Yaskawa INFORM job: X2_29-32(-90,180).JBI

/JOB
//NAME X2_29-32(-90,180)
//POS
///NPOS 301,301,301,19,0,0
///TOOL 0
///POSTYPE PULSE
///PULSE
C00000=-2000,-95440,-72516,0,38121,0
C00001=80443,-95440,-72516,46202,38121,-50067
C00002=52411,-63190,-65629,41206,65263,-51508
C00003=73087,-23788,-54178,20049,70640,-39353
C00004=137855,-58890,-63164,-50426,57117,-3007
C00005=121629,-1819,-23267,-32035,72941,-16834
C00006=120935,3126,-16373,-32060,71231,-16611
C00007=120668,5150,-13541,-32087,70531,-16512
C00008=120826,7275,-11699,-32150,70554,-16454
C00009=120668,5150,-13541,-32087,70531,-16512
C00010=120649,6560,-12069,-32112,70369,-16472
C00011=120645,6560,-10825,-32251,69714,-16277
C00012=120649,6560,-12069,-32112,70369,-16472
C00013=120913,4529,-14922,-32082,71075,-16573
C00014=121602,-429,-21862,-32048,72802,-16805
C00015=120074,-1541,-23154,-10906,71264,-22392
C00016=120462,3262,-16191,-11181,69532,-22093
C00017=120612,5232,-13331,-11295,68818,-21971
C00018=120770,7357,-11488,-11363,68799,-21912
C00019=120612,5232,-13331,-11295,68818,-21971
C00020=120702,6360,-12382,-11332,68826,-21940
C00021=120699,6356,-11141,-11388,68075,-21868
C00022=120702,6360,-12382,-11332,68826,-21940
C00023=120555,4389,-15254,-11219,69547,-22062
C00024=120172,-412,-22245,-10944,71297,-22361
C00025=119941,-49108,-60020,-12756,52739,-20459
C00026=119789,-74783,-79746,-11606,60570,-21449
C00027=121427,-115493,-86071,971,23186,-13
C00028=103613,-33005,-61039,35202,65094,22685
C00029=118652,-1130,-18887,50959,75871,22344
C00030=120065,3095,-12579,50928,73991,22034
C00031=120612,5858,-10323,50783,73711,22168
C00032=120794,7716,-8707,50742,73586,22192
C00033=120612,6719,-9575,50786,73699,22162
C00034=120612,6754,-8612,50907,73330,21953
C00035=120612,6719,-9575,50786,73699,22162
C00036=120164,4326,-11494,50910,73914,22043
C00037=118762,92,-17836,50934,75798,22362
C00038=120082,-2017,-23568,21020,76850,12939
C00039=120471,2786,-16617,21041,75059,12760
C00040=120621,6055,-13261,21027,74660,12744
C00041=120866,7545,-11965,20950,74569,12818
C00042=120698,6523,-12855,21003,74632,12768
C00043=120698,6506,-12245,21039,74273,12705
C00044=120698,6523,-12855,21003,74632,12768
C00045=120547,3972,-15593,21018,75020,12781
C00046=120163,-831,-22574,20994,76828,12964
C00047=120068,-2141,-23641,4094,79360,-4817
C00048=120458,2664,-16692,4000,77538,-4745
C00049=120609,5664,-13523,3960,77123,-4708
C00050=120915,7025,-12341,3868,77081,-4605
C00051=120609,5664,-13523,3960,77123,-4708
C00052=120609,5646,-12752,3962,76640,-4725
C00053=120609,5664,-13523,3960,77123,-4708
C00054=120559,4206,-15421,3970,77544,-4711
C00055=120175,-595,-22406,4061,79389,-4780
C00056=120687,14555,-20541,8533,86827,-5332
C00057=120686,13734,-18343,8544,85071,-5452
C00058=120482,15241,-16931,8603,84997,-5522
C00059=120827,14092,-17818,8504,84929,-5415
C00060=120926,18700,-11185,23232,84202,11400
C00061=120686,12663,-14714,25421,80171,12532
C00062=120686,13236,-17122,25321,81784,12881
C00063=103613,-33005,-61039,35202,65094,22685
C00064=121427,-115493,-86071,971,23186,-13
C00065=119789,-74783,-79746,-11606,60570,-21449
C00066=119941,-49108,-60020,-12756,52739,-20459
C00067=120686,14191,-18554,-15918,76373,-21593
C00068=120686,13500,-16249,-16032,74665,-21366
C00069=120864,13188,-15327,-16153,73998,-21217
C00070=120686,13025,-15397,-16089,73932,-21265
C00071=120685,13123,3553,-58384,63482,-21536
C00072=120685,12978,2576,-58170,63769,-21763
C00073=120685,12646,-109,-57582,64586,-22394
C00074=118042,2280,-28025,-21530,77386,-23855
C00075=119941,-49108,-60020,-12756,52739,-20459
C00076=119789,-74783,-79746,-11606,60570,-21449
C00077=121427,-115493,-86071,971,23186,-13
C00078=103613,-33005,-61039,35202,65094,22685
C00079=134099,37874,13933,30657,62495,29160
C00080=134100,37847,15487,30911,61654,28907
C00081=131666,39479,18748,33791,61688,27713
C00082=133865,38968,17694,31358,61081,28616
C00083=133702,39552,25338,55816,81533,5296
C00084=134106,38448,23823,57095,83317,3747
C00085=130543,37529,20923,57393,86199,3579
C00086=127607,4606,-13504,21031,60979,-34641
C00087=124532,-28339,-37080,-2656,37858,-63256
C00088=80443,-95440,-72516,46202,38121,-50067
C00089=628,-74499,-67639,57475,89722,-72456
C00090=-3643,-76224,-106676,-19950,71810,-76872
C00091=57022,-39792,-97587,14580,73098,-62715
C00092=77894,6609,-39652,10081,68656,-55583
C00093=79326,8848,-34628,9340,66588,-55287
C00094=79882,9812,-32559,9051,65763,-55166
C00095=80655,11957,-30643,8578,65611,-54918
C00096=79882,9812,-32559,9051,65763,-55166
C00097=80541,11612,-30977,8647,65649,-54954
C00098=80539,10894,-29907,8717,64633,-55031
C00099=80541,11612,-30977,8647,65649,-54954
C00100=79996,10638,-33064,8931,66478,-55073
C00101=78593,8374,-38132,9661,68553,-55366
C00102=77879,6415,-39661,10096,68566,-55596
C00103=79312,8664,-34633,9354,66499,-55298
C00104=79868,9631,-32562,9065,65674,-55178
C00105=80642,11778,-30647,8592,65523,-54929
C00106=79868,9631,-32562,9065,65674,-55178
C00107=80486,11377,-31039,8686,65573,-54978
C00108=80483,10662,-29965,8757,64557,-55056
C00109=80486,11377,-31039,8686,65573,-54978
C00110=79940,10400,-33127,8971,66401,-55097
C00111=78534,8129,-38197,9702,68474,-55392
C00112=80648,1920,-43069,8432,68075,-54741
C00113=82055,4328,-37962,7677,66061,-54418
C00114=82600,5356,-35863,7382,65258,-54288
C00115=83359,7582,-33929,6913,65152,-54039
C00116=82600,5356,-35863,7382,65258,-54288
C00117=83222,7216,-34336,6994,65225,-54082
C00118=83219,6503,-33246,7053,64194,-54145
C00119=83222,7216,-34336,6994,65225,-54082
C00120=82688,6183,-36451,7284,66032,-54210
C00121=81310,3762,-41594,8027,68053,-54528
C00122=103257,-17880,-58539,-5534,67057,-47481
C00123=104214,-14456,-52937,-6200,65440,-47084
C00124=104581,-13049,-50655,-6463,64788,-46925
C00125=105090,-10289,-48529,-6776,64935,-46761
C00126=104581,-13049,-50655,-6463,64788,-46925
C00127=105018,-10709,-48980,-6727,64992,-46789
C00128=105013,-11445,-47840,-6782,63918,-46728
C00129=105018,-10709,-48980,-6727,64992,-46789
C00130=104661,-12103,-51269,-6469,65653,-46947
C00131=103731,-15489,-56889,-5817,67299,-47340
C00132=80233,11979,-33534,13378,69985,-55632
C00133=80229,10556,-31784,13533,68226,-55836
C00134=80227,10062,-31089,13596,67561,-55913
C00135=85904,3072,-37201,10254,66968,-54061
C00136=91588,-2653,-41861,6857,66347,-52204
C00137=101831,-9955,-47602,630,65696,-48799
C00138=101534,-9526,-48387,809,66398,-48894
C00139=100861,-7653,-49935,1203,68321,-49097
C00140=80300,11336,-32181,3939,63811,-54132
C00141=80297,10024,-30348,4003,62013,-54196
C00142=80296,9591,-29657,4027,61367,-54219
C00143=80356,9906,-29534,3997,61454,-54195
C00144=80338,10281,-30338,3972,62137,-54177
C00145=80341,11605,-32161,3909,63935,-54114
C00146=57022,-39792,-97587,14580,73098,-62715
C00147=628,-74499,-67639,57475,89722,-72456
C00148=628,-74499,-67639,57475,89722,-72456
C00149=616,-75233,-71189,57531,90735,-71761
C00150=-3643,-76224,-106674,-19950,71813,-76873
C00151=42730,11015,-70691,38334,96086,-2936
C00152=63606,9545,-60534,45336,92087,16638
C00153=78956,5069,-41799,36523,82652,30708
C00154=79715,8164,-36018,36343,80767,30358
C00155=80007,9457,-33651,36288,80012,30216
C00156=80417,12097,-31285,36126,79775,30292
C00157=80007,9457,-33651,36288,80012,30216
C00158=80344,11698,-31669,36153,79828,30282
C00159=80337,10939,-30633,36254,78993,30001
C00160=80344,11698,-31669,36153,79828,30282
C00161=80059,10405,-34052,36203,80590,30428
C00162=79319,7312,-39869,36371,82488,30786
C00163=78994,5332,-41692,36502,82694,30736
C00164=79751,8420,-35912,36322,80808,30385
C00165=80043,9710,-33546,36267,80051,30242
C00166=80452,12349,-31177,36105,79813,30317
C00167=80043,9710,-33546,36267,80051,30242
C00168=80378,11838,-31671,36133,79874,30310
C00169=80371,11075,-30637,36233,79039,30029
C00170=80378,11838,-31671,36133,79874,30310
C00171=80093,10547,-34052,36183,80637,30456
C00172=79355,7462,-39866,36352,82536,30815
C00173=79090,5824,-41546,36452,82791,30803
C00174=79842,8894,-35770,36272,80900,30451
C00175=80133,10177,-33405,36216,80142,30307
C00176=80539,12815,-31031,36055,79902,30380
C00177=80133,10177,-33405,36216,80142,30307
C00178=80467,12378,-31515,36079,79989,30382
C00179=80461,11606,-30490,36178,79153,30101
C00180=80467,12378,-31515,36079,79989,30382
C00181=80184,11095,-33894,36130,80753,30529
C00182=79450,8031,-39703,36300,82657,30890
C00183=79130,5997,-41490,36432,82820,30827
C00184=79881,9061,-35715,36251,80928,30474
C00185=80171,10342,-33350,36196,80169,30330
C00186=80577,12980,-30974,36035,79928,30403
C00187=80171,10342,-33350,36196,80169,30330
C00188=80499,12601,-31443,36059,80034,30409
C00189=80493,11826,-30422,36158,79199,30129
C00190=80499,12601,-31443,36059,80034,30409
C00191=80216,11321,-33822,36110,80799,30556
C00192=79484,8265,-39628,36281,82705,30918
C00193=80360,13355,-34008,31162,79863,31191
C00194=80358,11846,-32319,31320,78301,30757
C00195=80218,11485,-31511,31450,77760,30555
C00196=80458,11751,-31298,31342,77685,30622
C00197=80398,12063,-32232,31297,78337,30782
C00198=80400,13577,-33916,31139,79899,31215
C00199=80289,11819,-32883,40833,82428,30239
C00200=80286,10439,-31086,40975,81039,29694
C00201=80075,10175,-30147,41122,80582,29428
C00202=80234,9688,-30441,41065,80463,29445
C00203=80245,10226,-31168,40996,81011,29666
C00204=80248,11601,-32971,40853,82401,30212
C00205=66712,19655,-58640,43457,90055,24381
C00206=33423,17994,-60377,60627,102988,19600
C00207=628,-74499,-67639,57475,89722,77289
C00208=111516,-94989,-87682,11539,41033,8318
C00209=107125,-12532,-46236,32676,64375,10703
C00210=119952,37605,6162,31233,75137,17424
C00211=120511,42562,14108,31354,72919,17016
C00212=120728,44654,17433,31427,72005,16841
C00213=120598,46946,19889,31526,71766,16719
C00214=120728,44654,17433,31427,72005,16841
C00215=120690,45788,18679,31469,71861,16784
C00216=120687,45721,19851,31594,71213,16595
C00217=120690,45788,18679,31469,71861,16784
C00218=120474,43679,15324,31394,72783,16962
C00219=119917,38688,7316,31265,75018,17376
C00220=121235,29127,929,10497,72605,22385
C00221=120892,33963,8709,10768,70384,22067
C00222=120760,35995,11952,10883,69467,21936
C00223=120625,38237,14258,10956,69222,21864
C00224=120760,35995,11952,10883,69467,21936
C00225=120657,37146,13206,10937,69303,21884
C00226=120654,37124,14427,10991,68554,21813
C00227=120657,37146,13206,10937,69303,21884
C00228=120788,35099,9935,10821,70230,22016
C00229=121127,30229,2096,10548,72470,22335
C00230=114017,-48711,-62992,16459,47417,13874
C00231=111516,-94989,-87682,11539,41033,8318
C00232=135207,-75469,-94215,-36619,68365,-13249
C00233=122507,12852,-43627,-17515,100315,-22769
C00234=122731,-562,-19309,-51196,76332,-22742
C00235=121309,3590,-13049,-51151,74446,-22427
C00236=120759,5312,-10468,-51156,73690,-22291
C00237=120602,7442,-8613,-51127,73573,-22309
C00238=120759,5312,-10468,-51156,73690,-22291
C00239=120666,6547,-9361,-51143,73609,-22295
C00240=120662,6597,-8073,-51308,73115,-22013
C00241=120666,6547,-9361,-51143,73609,-22295
C00242=121212,4820,-11958,-51134,74367,-22434
C00243=122622,659,-18251,-51172,76257,-22758
C00244=122507,10859,-42333,-17402,98575,-22516
C00245=121302,-1391,-23074,-21379,77148,-13095
C00246=120901,3377,-16122,-21398,75339,-12912
C00247=120747,5333,-13267,-21416,74597,-12833
C00248=120590,7459,-11416,-21370,74514,-12875
C00249=120747,5333,-13267,-21416,74597,-12833
C00250=120673,6521,-12221,-21396,74547,-12851
C00251=120670,6504,-10992,-21468,73832,-12721
C00252=120673,6521,-12221,-21396,74547,-12851
C00253=120826,4563,-15090,-21376,75296,-12931
C00254=121222,-206,-22073,-21354,77121,-13119
C00255=121314,-1652,-23262,-4485,79740,4708
C00256=120913,3117,-16316,-4391,77900,4639
C00257=120758,5074,-13462,-4356,77144,4613
C00258=120601,7199,-11615,-4311,77090,4561
C00259=120758,5074,-13462,-4356,77144,4613
C00260=120661,6618,-12165,-4328,77134,4580
C00261=120658,6600,-10936,-4339,76370,4606
C00262=120661,6618,-12165,-4328,77134,4580
C00263=120814,4660,-15035,-4362,77900,4605
C00264=121209,-107,-22019,-4454,79763,4672
C00265=120687,46979,12625,-8958,83453,5452
C00266=120687,46939,12852,-8960,83294,5464
C00267=121610,47264,14210,-9230,82736,5807
C00268=120687,46849,13873,-8967,82635,5512
C00269=120687,46629,18284,-25995,77833,-12130
C00270=120687,46348,16793,-25935,78533,-12285
C00271=120687,46750,14296,-25811,80109,-12635
C00272=133650,-5326,-40947,-35821,67459,-4738
C00273=126605,-79487,-84548,-34660,58331,-13454
C00274=111516,-94989,-87682,11539,41033,8318
C00275=114017,-48711,-62992,16459,47417,13874
C00276=117875,8541,-26754,15356,68464,18868
C00277=120687,46680,12303,15684,74586,21239
C00278=120687,46183,14573,15804,72993,21028
C00279=120687,45847,15503,15862,72274,20933
C00280=120687,45820,15711,15860,72146,20914
C00281=120686,46430,31549,51889,62431,21622
C00282=120686,46225,30262,51616,62867,21897
C00283=120686,45862,27317,50999,63909,22538
C00284=117875,8541,-26754,15356,68464,18868
C00285=114017,-48711,-62992,16459,47417,13874
C00286=111516,-94989,-87682,11539,41033,8318
C00287=126605,-79487,-84548,-34660,58331,-13454
C00288=133650,-5326,-40947,-35821,67459,-4738
C00289=107292,16878,-7589,-30401,64778,-29950
C00290=107291,16671,-4858,-30829,63228,-29495
C00291=107592,16882,-3413,-31166,62662,-29196
C00292=107321,17068,-3230,-31043,62555,-29280
C00293=107534,17274,4954,-56952,83139,-4906
C00294=107292,17076,4270,-57512,83951,-4302
C00295=107292,16842,1986,-57434,84665,-4798
C00296=118083,23141,-28416,-25698,115113,-5779
C00297=116334,-46006,-81849,-24511,89565,-1242
C00298=114916,-111361,-106536,-23911,54498,5439
C00299=628,-74499,-67639,57475,89722,77289
C00300=-2000,17994,-60377,0,102988,0
BC00000=30845,523905,744523
BC00001=125909,496171,117576
BC00002=171979,474261,96767
BC00003=199950,460958,84133
BC00004=289357,418436,43749
BC00005=289357,418436,43749
BC00006=289357,420740,43749
BC00007=289357,420740,43749
BC00008=289357,420740,43749
BC00009=289357,420740,43749
BC00010=289357,420740,43749
BC00011=289357,420740,43749
BC00012=289357,420740,43749
BC00013=289357,420740,43749
BC00014=289357,420740,43749
BC00015=275414,433755,78276
BC00016=275414,433755,78276
BC00017=275414,433755,78276
BC00018=275414,433755,78276
BC00019=275414,433755,78276
BC00020=275414,433755,78276
BC00021=275414,433755,78276
BC00022=275414,433755,78276
BC00023=275414,433755,78276
BC00024=275414,433755,78276
BC00025=275414,466967,78276
BC00026=275414,517660,78276
BC00027=159989,513142,117576
BC00028=134477,457942,17
BC00029=134477,457942,17
BC00030=134477,457942,17
BC00031=134477,457942,17
BC00032=134477,457942,17
BC00033=134477,457942,17
BC00034=134477,457942,17
BC00035=134477,457942,17
BC00036=134477,457942,17
BC00037=134477,457942,17
BC00038=119997,460424,63246
BC00039=119997,460424,63246
BC00040=119997,460424,63246
BC00041=119997,460424,63246
BC00042=119997,460424,63246
BC00043=119997,460424,63246
BC00044=119997,460424,63246
BC00045=119997,460424,63246
BC00046=119997,460424,63246
BC00047=143280,449314,87305
BC00048=143280,449314,87305
BC00049=143280,449314,87305
BC00050=143280,449314,87305
BC00051=143280,449314,87305
BC00052=143280,449314,87305
BC00053=143280,449314,87305
BC00054=143280,449314,87305
BC00055=143280,449314,87305
BC00056=160859,459195,5341
BC00057=159199,453961,5341
BC00058=159034,453443,5341
BC00059=154247,452737,5341
BC00060=124422,462638,5341
BC00061=121788,465826,5341
BC00062=123448,471060,5341
BC00063=134477,457942,17
BC00064=159989,513142,117576
BC00065=275414,517660,78276
BC00066=275414,466967,78276
BC00067=261614,447359,5341
BC00068=261319,441887,5341
BC00069=262619,439450,5341
BC00070=310184,431149,5341
BC00071=269021,423879,5341
BC00072=267544,425954,5341
BC00073=263853,431141,5341
BC00074=263853,431141,5341
BC00075=275414,466967,78276
BC00076=275414,517660,78276
BC00077=159989,513142,117576
BC00078=134477,457942,17
BC00079=177125,504351,5341
BC00080=175464,499117,5341
BC00081=174801,497234,5519
BC00082=160456,499532,5356
BC00083=152899,459984,5342
BC00084=154759,457798,5341
BC00085=160995,460631,5341
BC00086=160407,482802,71160
BC00087=159989,498475,117576
BC00088=125909,498475,117576
BC00089=97158,525533,426323
BC00090=199448,517843,1075137
BC00091=48431,468399,1061681
BC00092=196167,419409,1075139
BC00093=196167,419409,1075139
BC00094=196167,419409,1075139
BC00095=196167,419409,1075139
BC00096=196167,419409,1075139
BC00097=196167,419409,1075139
BC00098=196167,419409,1075139
BC00099=196167,419409,1075139
BC00100=196167,419409,1075139
BC00101=196167,419409,1075139
BC00102=139853,429285,1075139
BC00103=139853,429285,1075139
BC00104=139853,429285,1075139
BC00105=139853,429285,1075139
BC00106=139853,429285,1075139
BC00107=139853,429285,1075139
BC00108=139853,429285,1075139
BC00109=139853,429285,1075139
BC00110=139853,429285,1075139
BC00111=139853,429285,1075139
BC00112=1592,454839,1075139
BC00113=1592,454839,1075139
BC00114=1592,454839,1075139
BC00115=1592,454839,1075139
BC00116=1592,454839,1075139
BC00117=1592,454839,1075139
BC00118=1592,454839,1075139
BC00119=1592,454839,1075139
BC00120=1592,454839,1075139
BC00121=1592,454839,1075139
BC00122=1592,464839,1075139
BC00123=1592,464839,1075139
BC00124=1592,464839,1075139
BC00125=1592,464839,1075139
BC00126=1592,464839,1075139
BC00127=1592,464839,1075139
BC00128=1592,464839,1075139
BC00129=1592,464839,1075139
BC00130=1592,464839,1075139
BC00131=1592,464839,1075139
BC00132=12520,459695,1075139
BC00133=10860,454461,1075139
BC00134=10195,452368,1075139
BC00135=7188,455817,1075139
BC00136=4384,459034,1075139
BC00137=1592,464066,1075139
BC00138=1592,466159,1075139
BC00139=1592,471393,1075139
BC00140=125611,435762,1075139
BC00141=125317,430289,1075139
BC00142=125199,428100,1075139
BC00143=192322,416402,1075137
BC00144=192440,418591,1075139
BC00145=192735,424064,1075139
BC00146=48431,468399,1061681
BC00147=97158,523229,1005604
BC00148=97158,523229,842352
BC00149=97158,523229,900711
BC00150=199448,515539,1075136
BC00151=79980,453528,994842
BC00152=45336,436504,1043165
BC00153=33968,417480,1075139
BC00154=33968,417480,1075139
BC00155=33968,417480,1075139
BC00156=33968,417480,1075139
BC00157=33968,417480,1075139
BC00158=33968,417480,1075139
BC00159=33968,417480,1075139
BC00160=33968,417480,1075139
BC00161=33968,417480,1075139
BC00162=33968,417480,1075139
BC00163=90300,427260,1075139
BC00164=90300,427260,1075139
BC00165=90300,427260,1075139
BC00166=90300,427260,1075139
BC00167=90300,427260,1075139
BC00168=90300,427260,1075139
BC00169=90300,427260,1075139
BC00170=90300,427260,1075139
BC00171=90300,427260,1075139
BC00172=90300,427260,1075139
BC00173=237115,452564,1075139
BC00174=237115,452564,1075139
BC00175=237115,452564,1075139
BC00176=237115,452564,1075139
BC00177=237115,452564,1075139
BC00178=237115,452564,1075139
BC00179=237115,452564,1075139
BC00180=237115,452564,1075139
BC00181=237115,452564,1075139
BC00182=237115,452564,1075139
BC00183=294619,462466,1075139
BC00184=294619,462466,1075139
BC00185=294619,462466,1075139
BC00186=294619,462466,1075139
BC00187=294619,462466,1075139
BC00188=294619,462466,1075139
BC00189=294619,462466,1075139
BC00190=294619,462466,1075139
BC00191=294619,462466,1075139
BC00192=294619,462466,1075139
BC00193=217635,457409,1075139
BC00194=219331,452208,1075139
BC00195=220009,450128,1075139
BC00196=287154,461712,1075139
BC00197=286476,463793,1075139
BC00198=284781,468994,1075139
BC00199=104533,433695,1075139
BC00200=104861,428258,1075139
BC00201=104993,426083,1075139
BC00202=37847,414499,1075139
BC00203=37716,416674,1075139
BC00204=37387,422111,1075139
BC00205=32574,439916,986534
BC00206=32574,515576,986534
BC00207=97158,523229,426323
BC00208=147921,520101,17
BC00209=147921,478336,17
BC00210=147921,459959,17
BC00211=147921,459959,17
BC00212=147921,459959,17
BC00213=147921,459959,17
BC00214=147921,459959,17
BC00215=147921,459959,17
BC00216=147921,459959,17
BC00217=147921,459959,17
BC00218=147921,459959,17
BC00219=147921,459959,17
BC00220=158149,463458,58974
BC00221=158149,463458,58974
BC00222=158149,463458,58974
BC00223=158149,463458,58974
BC00224=158149,463458,58974
BC00225=158149,463458,58974
BC00226=158149,463458,58974
BC00227=158149,463458,58974
BC00228=158149,463458,58974
BC00229=158149,463458,58974
BC00230=154142,485648,35877
BC00231=147921,520101,17
BC00232=303952,516243,17
BC00233=303952,456764,17
BC00234=303952,456764,17
BC00235=303952,456764,17
BC00236=303952,456764,17
BC00237=303952,456764,17
BC00238=303952,456764,17
BC00239=303952,456764,17
BC00240=303952,456764,17
BC00241=303952,456764,17
BC00242=303952,456764,17
BC00243=303952,456764,17
BC00244=303952,456764,17
BC00245=317843,458872,70059
BC00246=317843,458872,70059
BC00247=317843,458872,70059
BC00248=317843,458872,70059
BC00249=317843,458872,70059
BC00250=317843,458872,70059
BC00251=317843,458872,70059
BC00252=317843,458872,70059
BC00253=317843,458872,70059
BC00254=317843,458872,70059
BC00255=294330,447356,94524
BC00256=294330,447356,94524
BC00257=294330,447356,94524
BC00258=294330,447356,94524
BC00259=294330,447356,94524
BC00260=294330,447356,94524
BC00261=294330,447356,94524
BC00262=294330,447356,94524
BC00263=294330,447356,94524
BC00264=294330,447356,94524
BC00265=276724,491586,17212
BC00266=278419,486385,17
BC00267=279097,484305,17
BC00268=283803,485104,17
BC00269=316748,496575,17
BC00270=316070,498656,17
BC00271=314375,503857,17
BC00272=314375,503857,17
BC00273=303952,516243,17
BC00274=147921,520101,17
BC00275=154142,485648,35877
BC00276=166900,482219,15684
BC00277=176256,479705,876
BC00278=176585,474268,17
BC00279=176716,472093,17
BC00280=127719,463629,15
BC00281=162006,459296,17
BC00282=163222,461417,17
BC00283=166262,466718,17
BC00284=166900,482219,15684
BC00285=154142,485648,35877
BC00286=147921,520101,17
BC00287=303952,516243,17
BC00288=314375,503857,17
BC00289=265194,481213,5341
BC00290=266889,476012,5341
BC00291=267568,473931,5341
BC00292=283248,476627,5341
BC00293=289731,434625,5341
BC00294=287455,434272,5341
BC00295=281194,437089,5341
BC00296=281194,437089,5341
BC00297=281194,437089,5341
BC00298=281194,437089,5341
BC00299=97158,523229,426323
BC00300=32574,515576,986534
EC00000=798156,-1296783
EC00001=798156,-1296783
EC00002=798156,-1296783
EC00003=798156,-1296783
EC00004=798156,-1296783
EC00005=798156,-1296783
EC00006=798156,-1296783
EC00007=798156,-1296783
EC00008=798156,-1296783
EC00009=798156,-1296783
EC00010=798156,-1296783
EC00011=798156,-1296783
EC00012=798156,-1296783
EC00013=798156,-1296783
EC00014=798156,-1296783
EC00015=798156,-1296783
EC00016=798156,-1296783
EC00017=798156,-1296783
EC00018=798156,-1296783
EC00019=798156,-1296783
EC00020=798156,-1296783
EC00021=798156,-1296783
EC00022=798156,-1296783
EC00023=798156,-1296783
EC00024=798156,-1296783
EC00025=798156,-1296783
EC00026=798156,-1296783
EC00027=798156,-1296783
EC00028=798156,-1296783
EC00029=798156,-1296783
EC00030=798156,-1296783
EC00031=798156,-1296783
EC00032=798156,-1296783
EC00033=798156,-1296783
EC00034=798156,-1296783
EC00035=798156,-1296783
EC00036=798156,-1296783
EC00037=798156,-1296783
EC00038=798156,-1296783
EC00039=798156,-1296783
EC00040=798156,-1296783
EC00041=798156,-1296783
EC00042=798156,-1296783
EC00043=798156,-1296783
EC00044=798156,-1296783
EC00045=798156,-1296783
EC00046=798156,-1296783
EC00047=798156,-1296783
EC00048=798156,-1296783
EC00049=798156,-1296783
EC00050=798156,-1296783
EC00051=798156,-1296783
EC00052=798156,-1296783
EC00053=798156,-1296783
EC00054=798156,-1296783
EC00055=798156,-1296783
EC00056=798156,-1296783
EC00057=798156,-1296783
EC00058=798156,-1296783
EC00059=798156,-1296783
EC00060=798156,-1296783
EC00061=798156,-1296783
EC00062=798156,-1296783
EC00063=798156,-1296783
EC00064=798156,-1296783
EC00065=798156,-1296783
EC00066=798156,-1296783
EC00067=798156,-1296783
EC00068=798156,-1296783
EC00069=798156,-1296783
EC00070=798156,-1296783
EC00071=798156,-1296783
EC00072=798156,-1296783
EC00073=798156,-1296783
EC00074=798156,-1296783
EC00075=798156,-1296783
EC00076=798156,-1296783
EC00077=798156,-1296783
EC00078=798156,-1296783
EC00079=798156,-1296783
EC00080=798156,-1296783
EC00081=798155,-1296783
EC00082=798156,-1296783
EC00083=798156,-1296783
EC00084=798156,-1296783
EC00085=798156,-1296783
EC00086=798153,-1296784
EC00087=798156,-1296783
EC00088=798156,-1296783
EC00089=798156,-1296783
EC00090=798156,-1296783
EC00091=798156,-1296783
EC00092=798156,-1296783
EC00093=798156,-1296783
EC00094=798156,-1296783
EC00095=798156,-1296783
EC00096=798156,-1296783
EC00097=798156,-1296783
EC00098=798156,-1296783
EC00099=798156,-1296783
EC00100=798156,-1296783
EC00101=798156,-1296783
EC00102=798156,-1296783
EC00103=798156,-1296783
EC00104=798156,-1296783
EC00105=798156,-1296783
EC00106=798156,-1296783
EC00107=798156,-1296783
EC00108=798156,-1296783
EC00109=798156,-1296783
EC00110=798156,-1296783
EC00111=798156,-1296783
EC00112=798156,-1296783
EC00113=798156,-1296783
EC00114=798156,-1296783
EC00115=798156,-1296783
EC00116=798156,-1296783
EC00117=798156,-1296783
EC00118=798156,-1296783
EC00119=798156,-1296783
EC00120=798156,-1296783
EC00121=798156,-1296783
EC00122=798156,-1296783
EC00123=798156,-1296783
EC00124=798156,-1296783
EC00125=798156,-1296783
EC00126=798156,-1296783
EC00127=798156,-1296783
EC00128=798156,-1296783
EC00129=798156,-1296783
EC00130=798156,-1296783
EC00131=798156,-1296783
EC00132=798156,-1296783
EC00133=798156,-1296783
EC00134=798156,-1296783
EC00135=798156,-1296783
EC00136=798156,-1296783
EC00137=798156,-1296783
EC00138=798156,-1296783
EC00139=798156,-1296783
EC00140=798156,-1296783
EC00141=798156,-1296783
EC00142=798156,-1296783
EC00143=798155,-1296783
EC00144=798156,-1296783
EC00145=798156,-1296783
EC00146=798156,-1296783
EC00147=798156,-1296783
EC00148=861577,-983133
EC00149=850885,-545682
EC00150=798154,-183829
EC00151=798156,-183832
EC00152=798156,-183832
EC00153=798156,-183832
EC00154=798156,-183832
EC00155=798156,-183832
EC00156=798156,-183832
EC00157=798156,-183832
EC00158=798156,-183832
EC00159=798156,-183832
EC00160=798156,-183832
EC00161=798156,-183832
EC00162=798156,-183832
EC00163=798156,-183832
EC00164=798156,-183832
EC00165=798156,-183832
EC00166=798156,-183832
EC00167=798156,-183832
EC00168=798156,-183832
EC00169=798156,-183832
EC00170=798156,-183832
EC00171=798156,-183832
EC00172=798156,-183832
EC00173=798156,-183832
EC00174=798156,-183832
EC00175=798156,-183832
EC00176=798156,-183832
EC00177=798156,-183832
EC00178=798156,-183832
EC00179=798156,-183832
EC00180=798156,-183832
EC00181=798156,-183832
EC00182=798156,-183832
EC00183=798156,-183832
EC00184=798156,-183832
EC00185=798156,-183832
EC00186=798156,-183832
EC00187=798156,-183832
EC00188=798156,-183832
EC00189=798156,-183832
EC00190=798156,-183832
EC00191=798156,-183832
EC00192=798156,-183832
EC00193=798156,-183832
EC00194=798156,-183832
EC00195=798156,-183832
EC00196=798156,-183832
EC00197=798156,-183832
EC00198=798156,-183832
EC00199=798156,-183832
EC00200=798156,-183832
EC00201=798156,-183832
EC00202=798156,-183832
EC00203=798156,-183832
EC00204=798156,-183832
EC00205=798156,-183832
EC00206=798156,-183832
EC00207=798156,-183832
EC00208=798156,-183832
EC00209=798156,-183832
EC00210=798156,-183832
EC00211=798156,-183832
EC00212=798156,-183832
EC00213=798156,-183832
EC00214=798156,-183832
EC00215=798156,-183832
EC00216=798156,-183832
EC00217=798156,-183832
EC00218=798156,-183832
EC00219=798156,-183832
EC00220=798156,-183832
EC00221=798156,-183832
EC00222=798156,-183832
EC00223=798156,-183832
EC00224=798156,-183832
EC00225=798156,-183832
EC00226=798156,-183832
EC00227=798156,-183832
EC00228=798156,-183832
EC00229=798156,-183832
EC00230=798156,-183832
EC00231=798156,-183832
EC00232=798156,-183832
EC00233=798156,-183832
EC00234=798156,-183832
EC00235=798156,-183832
EC00236=798156,-183832
EC00237=798156,-183832
EC00238=798156,-183832
EC00239=798156,-183832
EC00240=798156,-183832
EC00241=798156,-183832
EC00242=798156,-183832
EC00243=798156,-183832
EC00244=798156,-183832
EC00245=798156,-183832
EC00246=798156,-183832
EC00247=798156,-183832
EC00248=798156,-183832
EC00249=798156,-183832
EC00250=798156,-183832
EC00251=798156,-183832
EC00252=798156,-183832
EC00253=798156,-183832
EC00254=798156,-183832
EC00255=798156,-183832
EC00256=798156,-183832
EC00257=798156,-183832
EC00258=798156,-183832
EC00259=798156,-183832
EC00260=798156,-183832
EC00261=798156,-183832
EC00262=798156,-183832
EC00263=798156,-183832
EC00264=798156,-183832
EC00265=798156,-183832
EC00266=798156,-183832
EC00267=798156,-183832
EC00268=798156,-183832
EC00269=798156,-183832
EC00270=798156,-183832
EC00271=798156,-183832
EC00272=798156,-183832
EC00273=798156,-183832
EC00274=798156,-183832
EC00275=798156,-183832
EC00276=798156,-183832
EC00277=798156,-183832
EC00278=798156,-183832
EC00279=798156,-183832
EC00280=798155,-183831
EC00281=798156,-183832
EC00282=798156,-183832
EC00283=798156,-183832
EC00284=798156,-183832
EC00285=798156,-183832
EC00286=798156,-183832
EC00287=798156,-183832
EC00288=798156,-183832
EC00289=798156,-183832
EC00290=798156,-183832
EC00291=798156,-183832
EC00292=798156,-183832
EC00293=798156,-183832
EC00294=798156,-183832
EC00295=798156,-183832
EC00296=798156,-183832
EC00297=798156,-183832
EC00298=798156,-183832
EC00299=798156,-183832
EC00300=798156,-183832
///POSTYPE BASE
///RECTAN
///RCONF 0,0,0,0,1,0,0,0,0,0,0,0,0,0,0,0,0,0,0,0,0,0,0,0
P00006=2.006,1.622,-0.565,0.0000,0.0000,0.0000
P00021=0.073,2.058,-0.109,0.0000,0.0000,0.0000
P00022=2.006,1.622,-0.565,0.0000,0.0000,0.0000
///RCONF 0,0,0,0,0,0,0,0,0,0,0,0,0,0,0,0,0,0,0,0,0,0,0,0
P00023=-2.957,-4.083,2.762,0.0000,0.0000,0.0000
P00024=-1.466,-0.226,-0.419,0.0000,0.0000,0.0000
P00025=3.643,0.007,-2.585,0.0000,0.0000,0.0000
P00026=2.644,0.055,-2.583,0.0000,0.0000,0.0000
P00027=2.278,0.099,-4.210,0.0000,0.0000,0.0000
P00028=-1.778,-0.182,-2.050,0.0000,0.0000,0.0000
P00033=0.854,-1.099,3.047,0.0000,0.0000,0.0000
///RCONF 0,0,0,0,1,0,0,0,0,0,0,0,0,0,0,0,0,0,0,0,0,0,0,0
P00034=-8.151,9.743,-4.393,0.0000,0.0000,0.0000
///RCONF 0,0,0,0,0,0,0,0,0,0,0,0,0,0,0,0,0,0,0,0,0,0,0,0
P00035=0.390,-0.027,1.040,0.0000,0.0000,0.0000
P00036=-2.434,0.084,0.197,0.0000,0.0000,0.0000
P00041=-0.109,0.014,0.966,0.0000,0.0000,0.0000
P00042=-0.220,0.371,-0.613,0.0000,0.0000,0.0000
P00043=-0.179,-5.890,-3.227,0.0000,0.0000,0.0000
P00044=-8.560,-7.557,-5.232,0.0000,0.0000,0.0000
P00045=-8.836,-6.632,-1.438,0.0000,0.0000,0.0000
P00046=-7.725,-0.107,-2.878,0.0000,0.0000,0.0000
//INST
///DATE 2024/12/18 20:57
///ATTR SC,RW
///GROUP1 RB1,BS1
///GROUP2 ST1
NOP
'X2_29-32(-90,180)
MOVJ C00000 BC00000 VJ=100.00  +MOVJ EC00000 VJ=100.00
MOVJ C00001 BC00001 VJ=100.00  +MOVJ EC00001 VJ=100.00
MOVJ C00002 BC00002 VJ=100.00  +MOVJ EC00002 VJ=100.00
MOVJ C00003 BC00003 VJ=100.00  +MOVJ EC00003 VJ=100.00
MOVJ C00004 BC00004 VJ=100.00  +MOVJ EC00004 VJ=100.00
'Path S4862
SFTOF3D
MOVJ C00005 BC00005 VJ=100.00  +MOVJ EC00005 VJ=100.00
MOVL C00006 BC00006 V=800.0  +MOVJ EC00006 VJ=100.00
SMOVL C00007 BC00007 V=166.7  +MOVJ EC00007
SREFP 3 C00008 BC00008  +REFP EC00008
CALL JOB:SEARCH-R1-S13D
SET P042 P006
SFTON3D P042
SMOVL C00009 BC00009 V=166.7  +MOVJ EC00009
SMOVL C00010 BC00010 V=166.7  +MOVJ EC00010
SREFP 3 C00011 BC00011  +REFP EC00011
CALL JOB:SEARCH-R1-S13D
SET P042 P006
SFTON3D P042
SMOVL C00012 BC00012 V=166.7  +MOVJ EC00012
MOVL C00013 BC00013 V=800.0  +MOVJ EC00013 VJ=100.00
MOVL C00014 BC00014 V=1000.0  +MOVJ EC00014 VJ=100.00
'EndPath S4862
'Path S4863
SFTOF3D
MOVJ C00015 BC00015 VJ=100.00  +MOVJ EC00015 VJ=100.00
MOVL C00016 BC00016 V=800.0  +MOVJ EC00016 VJ=100.00
SMOVL C00017 BC00017 V=166.7  +MOVJ EC00017
SREFP 3 C00018 BC00018  +REFP EC00018
CALL JOB:SEARCH-R1-S13D
SET P041 P006
SFTON3D P041
SMOVL C00019 BC00019 V=166.7  +MOVJ EC00019
SMOVL C00020 BC00020 V=166.7  +MOVJ EC00020
SREFP 3 C00021 BC00021  +REFP EC00021
CALL JOB:SEARCH-R1-S13D
SET P041 P006
SFTON3D P041
SMOVL C00022 BC00022 V=166.7  +MOVJ EC00022
MOVL C00023 BC00023 V=800.0  +MOVJ EC00023 VJ=100.00
MOVL C00024 BC00024 V=1000.0  +MOVJ EC00024 VJ=100.00
'EndPath S4863
MOVJ C00025 BC00025 VJ=100.00  +MOVJ EC00025 VJ=100.00
MOVJ C00026 BC00026 VJ=100.00  +MOVJ EC00026 VJ=100.00
MOVJ C00027 BC00027 VJ=100.00  +MOVJ EC00027 VJ=100.00
MOVJ C00028 BC00028 VJ=100.00  +MOVJ EC00028 VJ=100.00
'Path S4864
SFTOF3D
MOVJ C00029 BC00029 VJ=100.00  +MOVJ EC00029 VJ=100.00
MOVL C00030 BC00030 V=800.0  +MOVJ EC00030 VJ=100.00
SMOVL C00031 BC00031 V=166.7  +MOVJ EC00031
SREFP 3 C00032 BC00032  +REFP EC00032
CALL JOB:SEARCH-R1-S13D
SET P045 P006
SFTON3D P045
SMOVL C00033 BC00033 V=166.7  +MOVJ EC00033
SREFP 3 C00034 BC00034  +REFP EC00034
CALL JOB:SEARCH-R1-S13D
SET P045 P006
SFTON3D P045
SMOVL C00035 BC00035 V=166.7  +MOVJ EC00035
MOVL C00036 BC00036 V=800.0  +MOVJ EC00036 VJ=100.00
MOVL C00037 BC00037 V=1000.0  +MOVJ EC00037 VJ=100.00
'EndPath S4864
'Path S4231
SFTOF3D
MOVJ C00038 BC00038 VJ=100.00  +MOVJ EC00038 VJ=100.00
MOVL C00039 BC00039 V=800.0  +MOVJ EC00039 VJ=100.00
SMOVL C00040 BC00040 V=166.7  +MOVJ EC00040
SREFP 3 C00041 BC00041  +REFP EC00041
CALL JOB:SEARCH-R1-S13D
SET P022 P006
SFTON3D P022
SMOVL C00042 BC00042 V=166.7  +MOVJ EC00042
SREFP 3 C00043 BC00043  +REFP EC00043
CALL JOB:SEARCH-R1-S13D
SET P022 P006
SFTON3D P022
SMOVL C00044 BC00044 V=166.7  +MOVJ EC00044
MOVL C00045 BC00045 V=800.0  +MOVJ EC00045 VJ=100.00
MOVL C00046 BC00046 V=1000.0  +MOVJ EC00046 VJ=100.00
'EndPath S4231
'Path S4232
SFTOF3D
MOVJ C00047 BC00047 VJ=100.00  +MOVJ EC00047 VJ=100.00
MOVL C00048 BC00048 V=800.0  +MOVJ EC00048 VJ=100.00
SMOVL C00049 BC00049 V=166.7  +MOVJ EC00049
SREFP 3 C00050 BC00050  +REFP EC00050
CALL JOB:SEARCH-R1-S13D
SET P021 P006
SFTON3D P021
SMOVL C00051 BC00051 V=166.7  +MOVJ EC00051
SREFP 3 C00052 BC00052  +REFP EC00052
CALL JOB:SEARCH-R1-S13D
SET P021 P006
SFTON3D P021
SMOVL C00053 BC00053 V=166.7  +MOVJ EC00053
MOVL C00054 BC00054 V=800.0  +MOVJ EC00054 VJ=100.00
MOVL C00055 BC00055 V=1000.0  +MOVJ EC00055 VJ=100.00
'EndPath S4232
'Path W4886
SFTOF3D
SFTON3D P021
MOVJ C00056 BC00056 VJ=100.00  +MOVJ EC00056 VJ=100.00
SMOVL C00057 BC00057 V=800.0  +MOVJ EC00057
SMOVL C00058 BC00058 V=150.0 PL=0  +MOVJ EC00058
MACRO1 MJ#(0) ARGF6
ARCON
SMOVL C00059 BC00059 V=8.3  +MOVJ EC00059
SFTON3D P022
SMOVL C00060 BC00060 V=8.3  +MOVJ EC00060
ARCOF
SMOVL C00061 BC00061 V=800.0  +MOVJ EC00061
SMOVL C00062 BC00062 V=1000.0  +MOVJ EC00062
SFTOF3D
'EndPath W4886
MOVJ C00063 BC00063 VJ=100.00  +MOVJ EC00063 VJ=100.00
MOVJ C00064 BC00064 VJ=100.00  +MOVJ EC00064 VJ=100.00
MOVJ C00065 BC00065 VJ=100.00  +MOVJ EC00065 VJ=100.00
MOVJ C00066 BC00066 VJ=100.00  +MOVJ EC00066 VJ=100.00
'Path W4887
SFTOF3D
SFTON3D P041
MOVJ C00067 BC00067 VJ=100.00  +MOVJ EC00067 VJ=100.00
SMOVL C00068 BC00068 V=800.0  +MOVJ EC00068
SMOVL C00069 BC00069 V=150.0 PL=0  +MOVJ EC00069
ARCON
SMOVL C00070 BC00070 V=8.3  +MOVJ EC00070
SFTON3D P042
SMOVL C00071 BC00071 V=8.3  +MOVJ EC00071
ARCOF
SMOVL C00072 BC00072 V=800.0  +MOVJ EC00072
SMOVL C00073 BC00073 V=1000.0  +MOVJ EC00073
SFTOF3D
'EndPath W4887
MOVJ C00074 BC00074 VJ=100.00  +MOVJ EC00074 VJ=100.00
MOVJ C00075 BC00075 VJ=100.00  +MOVJ EC00075 VJ=100.00
MOVJ C00076 BC00076 VJ=100.00  +MOVJ EC00076 VJ=100.00
MOVJ C00077 BC00077 VJ=100.00  +MOVJ EC00077 VJ=100.00
MOVJ C00078 BC00078 VJ=100.00  +MOVJ EC00078 VJ=100.00
'Path W4887
SFTOF3D
SFTON3D P045
MOVJ C00079 BC00079 VJ=100.00  +MOVJ EC00079 VJ=100.00
SMOVL C00080 BC00080 V=800.0  +MOVJ EC00080
SMOVL C00081 BC00081 V=150.0 PL=0  +MOVJ EC00081
ARCON
SMOVL C00082 BC00082 V=8.3  +MOVJ EC00082
SMOVL C00083 BC00083 V=8.3  +MOVJ EC00083
ARCOF
SMOVL C00084 BC00084 V=800.0  +MOVJ EC00084
SMOVL C00085 BC00085 V=1000.0  +MOVJ EC00085
SFTOF3D
MOVJ C00086 BC00086 VJ=20.00  +MOVJ EC00086 VJ=20.00
'EndPath W4887
MOVJ C00087 BC00087 VJ=100.00  +MOVJ EC00087 VJ=100.00
MOVJ C00088 BC00088 VJ=100.00  +MOVJ EC00088 VJ=100.00
MOVJ C00089 BC00089 VJ=100.00  +MOVJ EC00089 VJ=100.00
'R-L Trip
MOVJ C00090 BC00090 VJ=100.00  +MOVJ EC00090 VJ=100.00
CALL JOB:CLEAN-R1_KM_NEW
'WireCut
MOVJ C00091 BC00091 VJ=100.00  +MOVJ EC00091 VJ=100.00
'Path S4234
SFTOF3D
MOVJ C00092 BC00092 VJ=100.00  +MOVJ EC00092 VJ=100.00
MOVL C00093 BC00093 V=800.0  +MOVJ EC00093 VJ=100.00
SMOVL C00094 BC00094 V=166.7  +MOVJ EC00094
SREFP 3 C00095 BC00095  +REFP EC00095
CALL JOB:SEARCH-R1-S13D
SET P034 P006
SFTON3D P034
SMOVL C00096 BC00096 V=166.7  +MOVJ EC00096
SMOVL C00097 BC00097 V=166.7  +MOVJ EC00097
SREFP 3 C00098 BC00098  +REFP EC00098
CALL JOB:SEARCH-R1-S13D
SET P034 P006
SFTON3D P034
SMOVL C00099 BC00099 V=166.7  +MOVJ EC00099
MOVL C00100 BC00100 V=800.0  +MOVJ EC00100 VJ=100.00
MOVL C00101 BC00101 V=1000.0  +MOVJ EC00101 VJ=100.00
'EndPath S4234
'Path S4235
SFTOF3D
MOVJ C00102 BC00102 VJ=100.00  +MOVJ EC00102 VJ=100.00
MOVL C00103 BC00103 V=800.0  +MOVJ EC00103 VJ=100.00
SMOVL C00104 BC00104 V=166.7  +MOVJ EC00104
SREFP 3 C00105 BC00105  +REFP EC00105
CALL JOB:SEARCH-R1-S13D
SET P033 P006
SFTON3D P033
SMOVL C00106 BC00106 V=166.7  +MOVJ EC00106
SMOVL C00107 BC00107 V=166.7  +MOVJ EC00107
SREFP 3 C00108 BC00108  +REFP EC00108
CALL JOB:SEARCH-R1-S13D
SET P033 P006
SFTON3D P033
SMOVL C00109 BC00109 V=166.7  +MOVJ EC00109
MOVL C00110 BC00110 V=800.0  +MOVJ EC00110 VJ=100.00
MOVL C00111 BC00111 V=1000.0  +MOVJ EC00111 VJ=100.00
'EndPath S4235
'Path S4236
SFTOF3D
MOVJ C00112 BC00112 VJ=100.00  +MOVJ EC00112 VJ=100.00
MOVL C00113 BC00113 V=800.0  +MOVJ EC00113 VJ=100.00
SMOVL C00114 BC00114 V=166.7  +MOVJ EC00114
SREFP 3 C00115 BC00115  +REFP EC00115
CALL JOB:SEARCH-R1-S13D
SET P024 P006
SFTON3D P024
SMOVL C00116 BC00116 V=166.7  +MOVJ EC00116
SMOVL C00117 BC00117 V=166.7  +MOVJ EC00117
SREFP 3 C00118 BC00118  +REFP EC00118
CALL JOB:SEARCH-R1-S13D
SET P024 P006
SFTON3D P024
SMOVL C00119 BC00119 V=166.7  +MOVJ EC00119
MOVL C00120 BC00120 V=800.0  +MOVJ EC00120 VJ=100.00
MOVL C00121 BC00121 V=1000.0  +MOVJ EC00121 VJ=100.00
'EndPath S4236
'Path S4237
SFTOF3D
MOVJ C00122 BC00122 VJ=100.00  +MOVJ EC00122 VJ=100.00
MOVL C00123 BC00123 V=800.0  +MOVJ EC00123 VJ=100.00
SMOVL C00124 BC00124 V=166.7  +MOVJ EC00124
SREFP 3 C00125 BC00125  +REFP EC00125
CALL JOB:SEARCH-R1-S13D
SET P023 P006
SFTON3D P023
SMOVL C00126 BC00126 V=166.7  +MOVJ EC00126
SMOVL C00127 BC00127 V=166.7  +MOVJ EC00127
SREFP 3 C00128 BC00128  +REFP EC00128
CALL JOB:SEARCH-R1-S13D
SET P023 P006
SFTON3D P023
SMOVL C00129 BC00129 V=166.7  +MOVJ EC00129
MOVL C00130 BC00130 V=800.0  +MOVJ EC00130 VJ=100.00
MOVL C00131 BC00131 V=1000.0  +MOVJ EC00131 VJ=100.00
'EndPath S4237
'nowe
'Path W4903
SFTOF3D
SFTON3D P024
MOVJ C00132 BC00132 VJ=100.00  +MOVJ EC00132 VJ=100.00
SMOVL C00133 BC00133 V=800.0  +MOVJ EC00133
SMOVL C00134 BC00134 V=150.0 PL=0  +MOVJ EC00134
MACRO1 MJ#(0) ARGF14
ARCON
SMOVL C00135 BC00135 V=9.2  +MOVJ EC00135
SFTON3D P023
SMOVL C00136 BC00136 V=9.2  +MOVJ EC00136
SMOVL C00137 BC00137 V=9.2  +MOVJ EC00137
ARCOF
SMOVL C00138 BC00138 V=800.0  +MOVJ EC00138
SMOVL C00139 BC00139 V=1000.0  +MOVJ EC00139
SFTOF3D
'EndPath W4903
'Path W4906
SFTOF3D
SFTON3D P033
MOVJ C00140 BC00140 VJ=100.00  +MOVJ EC00140 VJ=100.00
SMOVL C00141 BC00141 V=800.0  +MOVJ EC00141
SMOVL C00142 BC00142 V=150.0 PL=0  +MOVJ EC00142
ARCON
SFTON3D P034
SMOVL C00143 BC00143 V=10.7  +MOVJ EC00143
ARCOF
SMOVL C00144 BC00144 V=800.0  +MOVJ EC00144
SMOVL C00145 BC00145 V=1000.0  +MOVJ EC00145
SFTOF3D
'EndPath W4906
MOVJ C00146 BC00146 VJ=100.00  +MOVJ EC00146 VJ=100.00
'WireCut
MOVJ C00147 BC00147 VJ=100.00  +MOVJ EC00147 VJ=100.00
MOVJ C00148 BC00148 VJ=100.00  +MOVJ EC00148 VJ=100.00
MOVJ C00149 BC00149 VJ=100.00  +MOVJ EC00149 VJ=100.00
MOVJ C00150 BC00150 VJ=100.00  +MOVJ EC00150 VJ=100.00
CALL JOB:CLEAN-R1_KM_NEW
MOVJ C00151 BC00151 VJ=100.00  +MOVJ EC00151 VJ=100.00
MOVJ C00152 BC00152 VJ=100.00  +MOVJ EC00152 VJ=100.00
'L-R Trip
'Path S4249
SFTOF3D
MOVJ C00153 BC00153 VJ=100.00  +MOVJ EC00153 VJ=100.00
MOVL C00154 BC00154 V=800.0  +MOVJ EC00154 VJ=100.00
SMOVL C00155 BC00155 V=166.7  +MOVJ EC00155
SREFP 3 C00156 BC00156  +REFP EC00156
CALL JOB:SEARCH-R1-S13D
SET P036 P006
SFTON3D P036
SMOVL C00157 BC00157 V=166.7  +MOVJ EC00157
SMOVL C00158 BC00158 V=166.7  +MOVJ EC00158
SREFP 3 C00159 BC00159  +REFP EC00159
CALL JOB:SEARCH-R1-S13D
SET P036 P006
SFTON3D P036
SMOVL C00160 BC00160 V=166.7  +MOVJ EC00160
MOVL C00161 BC00161 V=800.0  +MOVJ EC00161 VJ=100.00
MOVL C00162 BC00162 V=1000.0  +MOVJ EC00162 VJ=100.00
'EndPath S4249
'Path S4250
SFTOF3D
MOVJ C00163 BC00163 VJ=100.00  +MOVJ EC00163 VJ=100.00
MOVL C00164 BC00164 V=800.0  +MOVJ EC00164 VJ=100.00
SMOVL C00165 BC00165 V=166.7  +MOVJ EC00165
SREFP 3 C00166 BC00166  +REFP EC00166
CALL JOB:SEARCH-R1-S13D
SET P035 P006
SFTON3D P035
SMOVL C00167 BC00167 V=166.7  +MOVJ EC00167
SMOVL C00168 BC00168 V=166.7  +MOVJ EC00168
SREFP 3 C00169 BC00169  +REFP EC00169
CALL JOB:SEARCH-R1-S13D
SET P035 P006
SFTON3D P035
SMOVL C00170 BC00170 V=166.7  +MOVJ EC00170
MOVL C00171 BC00171 V=800.0  +MOVJ EC00171 VJ=100.00
MOVL C00172 BC00172 V=1000.0  +MOVJ EC00172 VJ=100.00
'EndPath S4250
'Path S4251
SFTOF3D
MOVJ C00173 BC00173 VJ=100.00  +MOVJ EC00173 VJ=100.00
MOVL C00174 BC00174 V=800.0  +MOVJ EC00174 VJ=100.00
SMOVL C00175 BC00175 V=166.7  +MOVJ EC00175
SREFP 3 C00176 BC00176  +REFP EC00176
CALL JOB:SEARCH-R1-S13D
SET P026 P006
SFTON3D P026
SMOVL C00177 BC00177 V=166.7  +MOVJ EC00177
SMOVL C00178 BC00178 V=166.7  +MOVJ EC00178
SREFP 3 C00179 BC00179  +REFP EC00179
CALL JOB:SEARCH-R1-S13D
SET P026 P006
SFTON3D P026
SMOVL C00180 BC00180 V=166.7  +MOVJ EC00180
MOVL C00181 BC00181 V=800.0  +MOVJ EC00181 VJ=100.00
MOVL C00182 BC00182 V=1000.0  +MOVJ EC00182 VJ=100.00
'EndPath S4251
'Path S4252
SFTOF3D
MOVJ C00183 BC00183 VJ=100.00  +MOVJ EC00183 VJ=100.00
MOVL C00184 BC00184 V=800.0  +MOVJ EC00184 VJ=100.00
SMOVL C00185 BC00185 V=166.7  +MOVJ EC00185
SREFP 3 C00186 BC00186  +REFP EC00186
CALL JOB:SEARCH-R1-S13D
SET P025 P006
SFTON3D P025
SMOVL C00187 BC00187 V=166.7  +MOVJ EC00187
SMOVL C00188 BC00188 V=166.7  +MOVJ EC00188
SREFP 3 C00189 BC00189  +REFP EC00189
CALL JOB:SEARCH-R1-S13D
SET P025 P006
SFTON3D P025
SMOVL C00190 BC00190 V=166.7  +MOVJ EC00190
MOVL C00191 BC00191 V=800.0  +MOVJ EC00191 VJ=100.00
MOVL C00192 BC00192 V=1000.0  +MOVJ EC00192 VJ=100.00
'EndPath S4252
'Path W4907
SFTOF3D
SFTON3D P026
MOVJ C00193 BC00193 VJ=100.00  +MOVJ EC00193 VJ=100.00
SMOVL C00194 BC00194 V=800.0  +MOVJ EC00194
SMOVL C00195 BC00195 V=150.0 PL=0  +MOVJ EC00195
ARCON
SFTON3D P025
SMOVL C00196 BC00196 V=11.7  +MOVJ EC00196
ARCOF
SMOVL C00197 BC00197 V=800.0  +MOVJ EC00197
SMOVL C00198 BC00198 V=1000.0  +MOVJ EC00198
SFTOF3D
'EndPath W4907
'Path W4908
SFTOF3D
SFTON3D P035
MOVJ C00199 BC00199 VJ=100.00  +MOVJ EC00199 VJ=100.00
SMOVL C00200 BC00200 V=800.0  +MOVJ EC00200
SMOVL C00201 BC00201 V=150.0 PL=0  +MOVJ EC00201
ARCON
SFTON3D P036
SMOVL C00202 BC00202 V=11.7  +MOVJ EC00202
ARCOF
SMOVL C00203 BC00203 V=800.0  +MOVJ EC00203
SMOVL C00204 BC00204 V=1000.0  +MOVJ EC00204
SFTOF3D
'EndPath W4908
MOVJ C00205 BC00205 VJ=100.00  +MOVJ EC00205 VJ=100.00
MOVJ C00206 BC00206 VJ=100.00  +MOVJ EC00206 VJ=100.00
CALL JOB:CLEAN-R1_KM_NEW
MOVJ C00207 BC00207 VJ=100.00  +MOVJ EC00207 VJ=100.00
MOVJ C00208 BC00208 VJ=100.00  +MOVJ EC00208 VJ=100.00
MOVJ C00209 BC00209 VJ=100.00  +MOVJ EC00209 VJ=100.00
'Path S4888
SFTOF3D
MOVJ C00210 BC00210 VJ=100.00  +MOVJ EC00210 VJ=100.00
MOVL C00211 BC00211 V=800.0  +MOVJ EC00211 VJ=100.00
SMOVL C00212 BC00212 V=166.7  +MOVJ EC00212
SREFP 3 C00213 BC00213  +REFP EC00213
CALL JOB:SEARCH-R1-S13D
SET P044 P006
SFTON3D P044
SMOVL C00214 BC00214 V=166.7  +MOVJ EC00214
SMOVL C00215 BC00215 V=166.7  +MOVJ EC00215
SREFP 3 C00216 BC00216  +REFP EC00216
CALL JOB:SEARCH-R1-S13D
SET P044 P006
SFTON3D P044
SMOVL C00217 BC00217 V=166.7  +MOVJ EC00217
MOVL C00218 BC00218 V=800.0  +MOVJ EC00218 VJ=100.00
MOVL C00219 BC00219 V=1000.0  +MOVJ EC00219 VJ=100.00
'EndPath S4888
'Path S4889
SFTOF3D
MOVJ C00220 BC00220 VJ=100.00  +MOVJ EC00220 VJ=100.00
MOVL C00221 BC00221 V=800.0  +MOVJ EC00221 VJ=100.00
SMOVL C00222 BC00222 V=166.7  +MOVJ EC00222
SREFP 3 C00223 BC00223  +REFP EC00223
CALL JOB:SEARCH-R1-S13D
SET P043 P006
SFTON3D P043
SMOVL C00224 BC00224 V=166.7  +MOVJ EC00224
SMOVL C00225 BC00225 V=166.7  +MOVJ EC00225
SREFP 3 C00226 BC00226  +REFP EC00226
CALL JOB:SEARCH-R1-S13D
SET P043 P006
SFTON3D P043
SMOVL C00227 BC00227 V=166.7  +MOVJ EC00227
MOVL C00228 BC00228 V=800.0  +MOVJ EC00228 VJ=100.00
MOVL C00229 BC00229 V=1000.0  +MOVJ EC00229 VJ=100.00
'EndPath S4889
MOVJ C00230 BC00230 VJ=100.00  +MOVJ EC00230 VJ=100.00
MOVJ C00231 BC00231 VJ=100.00  +MOVJ EC00231 VJ=100.00
MOVJ C00232 BC00232 VJ=100.00  +MOVJ EC00232 VJ=100.00
MOVJ C00233 BC00233 VJ=100.00  +MOVJ EC00233 VJ=100.00
'Path S4899
SFTOF3D
MOVJ C00234 BC00234 VJ=100.00  +MOVJ EC00234 VJ=100.00
MOVL C00235 BC00235 V=800.0  +MOVJ EC00235 VJ=100.00
SMOVL C00236 BC00236 V=166.7  +MOVJ EC00236
SREFP 3 C00237 BC00237  +REFP EC00237
CALL JOB:SEARCH-R1-S13D
SET P046 P006
SFTON3D P046
SMOVL C00238 BC00238 V=166.7  +MOVJ EC00238
SMOVL C00239 BC00239 V=166.7  +MOVJ EC00239
SREFP 3 C00240 BC00240  +REFP EC00240
CALL JOB:SEARCH-R1-S13D
SET P046 P006
SFTON3D P046
SMOVL C00241 BC00241 V=166.7  +MOVJ EC00241
MOVL C00242 BC00242 V=800.0  +MOVJ EC00242 VJ=100.00
MOVL C00243 BC00243 V=1000.0  +MOVJ EC00243 VJ=100.00
'EndPath S4899
MOVJ C00244 BC00244 VJ=100.00  +MOVJ EC00244 VJ=100.00
'Path S4888
SFTOF3D
MOVJ C00245 BC00245 VJ=100.00  +MOVJ EC00245 VJ=100.00
MOVL C00246 BC00246 V=800.0  +MOVJ EC00246 VJ=100.00
SMOVL C00247 BC00247 V=166.7  +MOVJ EC00247
SREFP 3 C00248 BC00248  +REFP EC00248
CALL JOB:SEARCH-R1-S13D
SET P028 P006
SFTON3D P028
SMOVL C00249 BC00249 V=166.7  +MOVJ EC00249
SMOVL C00250 BC00250 V=166.7  +MOVJ EC00250
SREFP 3 C00251 BC00251  +REFP EC00251
CALL JOB:SEARCH-R1-S13D
SET P028 P006
SFTON3D P028
SMOVL C00252 BC00252 V=166.7  +MOVJ EC00252
MOVL C00253 BC00253 V=800.0  +MOVJ EC00253 VJ=100.00
MOVL C00254 BC00254 V=1000.0  +MOVJ EC00254 VJ=100.00
'EndPath S4888
'Path S4889
SFTOF3D
MOVJ C00255 BC00255 VJ=100.00  +MOVJ EC00255 VJ=100.00
MOVL C00256 BC00256 V=800.0  +MOVJ EC00256 VJ=100.00
SMOVL C00257 BC00257 V=166.7  +MOVJ EC00257
SREFP 3 C00258 BC00258  +REFP EC00258
CALL JOB:SEARCH-R1-S13D
SET P027 P006
SFTON3D P027
SMOVL C00259 BC00259 V=166.7  +MOVJ EC00259
SMOVL C00260 BC00260 V=166.7  +MOVJ EC00260
SREFP 3 C00261 BC00261  +REFP EC00261
CALL JOB:SEARCH-R1-S13D
SET P027 P006
SFTON3D P027
SMOVL C00262 BC00262 V=166.7  +MOVJ EC00262
MOVL C00263 BC00263 V=800.0  +MOVJ EC00263 VJ=100.00
MOVL C00264 BC00264 V=1000.0  +MOVJ EC00264 VJ=100.00
'EndPath S4889
'Path W4890
SFTOF3D
SFTON3D P027
MOVJ C00265 BC00265 VJ=100.00  +MOVJ EC00265 VJ=100.00
SMOVL C00266 BC00266 V=800.0  +MOVJ EC00266
SMOVL C00267 BC00267 V=150.0 PL=0  +MOVJ EC00267
MACRO1 MJ#(0) ARGF6
ARCON
SMOVL C00268 BC00268 V=6.7  +MOVJ EC00268
SFTON3D P028
SMOVL C00269 BC00269 V=10.0  +MOVJ EC00269
ARCOF
SMOVL C00270 BC00270 V=800.0  +MOVJ EC00270
SMOVL C00271 BC00271 V=1000.0  +MOVJ EC00271
SFTOF3D
'EndPath W4890
MOVJ C00272 BC00272 VJ=100.00  +MOVJ EC00272 VJ=100.00
MOVJ C00273 BC00273 VJ=100.00  +MOVJ EC00273 VJ=100.00
MOVJ C00274 BC00274 VJ=100.00  +MOVJ EC00274 VJ=100.00
MOVJ C00275 BC00275 VJ=100.00  +MOVJ EC00275 VJ=100.00
MOVJ C00276 BC00276 VJ=100.00  +MOVJ EC00276 VJ=100.00
'Path W4900
SFTOF3D
SFTON3D P043
MOVJ C00277 BC00277 VJ=100.00  +MOVJ EC00277 VJ=100.00
SMOVL C00278 BC00278 V=800.0  +MOVJ EC00278
SMOVL C00279 BC00279 V=150.0 PL=0  +MOVJ EC00279
MACRO1 MJ#(0) ARGF14
ARCON
SFTON3D P044
SMOVL C00280 BC00280 V=10.0  +MOVJ EC00280
SMOVL C00281 BC00281 V=10.0  +MOVJ EC00281
ARCOF
SMOVL C00282 BC00282 V=800.0  +MOVJ EC00282
SMOVL C00283 BC00283 V=1000.0  +MOVJ EC00283
SFTOF3D
'EndPath W4900
MOVJ C00284 BC00284 VJ=100.00  +MOVJ EC00284 VJ=100.00
MOVJ C00285 BC00285 VJ=100.00  +MOVJ EC00285 VJ=100.00
MOVJ C00286 BC00286 VJ=100.00  +MOVJ EC00286 VJ=100.00
MOVJ C00287 BC00287 VJ=100.00  +MOVJ EC00287 VJ=100.00
MOVJ C00288 BC00288 VJ=100.00  +MOVJ EC00288 VJ=100.00
'Path W4898
SFTOF3D
SFTON3D P046
MOVJ C00289 BC00289 VJ=100.00  +MOVJ EC00289 VJ=100.00
SMOVL C00290 BC00290 V=800.0  +MOVJ EC00290
SMOVL C00291 BC00291 V=150.0 PL=0  +MOVJ EC00291
ARCON
SMOVL C00292 BC00292 V=10.0  +MOVJ EC00292
SMOVL C00293 BC00293 V=10.0  +MOVJ EC00293
ARCOF
SMOVL C00294 BC00294 V=800.0  +MOVJ EC00294
SMOVL C00295 BC00295 V=1000.0  +MOVJ EC00295
SFTOF3D
'EndPath W4898
MOVJ C00296 BC00296 VJ=100.00  +MOVJ EC00296 VJ=100.00
MOVJ C00297 BC00297 VJ=100.00  +MOVJ EC00297 VJ=100.00
MOVJ C00298 BC00298 VJ=100.00  +MOVJ EC00298 VJ=100.00
MOVJ C00299 BC00299 VJ=100.00  +MOVJ EC00299 VJ=100.00
MOVJ C00300 BC00300 VJ=100.00  +MOVJ EC00300 VJ=100.00
END
